TYPE ST_elpriserJustNu24Timmar :
STRUCT
	elpriserTimme: ARRAY[1..23] OF ST_elpriserTimme;
	
END_STRUCT
END_TYPE

(* stored: Version 1.1.0.1, ProductVersion 3.1.4024.12
   DUT ST_elpriserJustNu24Timmar: Id {4c18c218-d0fe-4dcb-b5f9-123c511ce7d3} *)
